PROGRAM INTERNAL PRG_TEST_FB_MANUALCONTROLLER
VAR
	bEnableTests : BOOL;

	bInitDone 			: BOOL;
	fbManualController 	: FB_ManualController;
	fbDevValve 			: FB_DevValve;
END_VAR

IF bEnableTests THEN
	IF NOT bInitDone THEN
		bInitDone := TRUE;
		fbDevValve.Init(
			nId := 1,
			nParentId := 0,
			eResetState := E_ValveResetState.Res_Idle,
			eSafeState := E_ValveResetState.Res_Idle
		);
	END_IF
	
	fbManualController();
	fbDevValve(
		refFbManualCtrl	:= fbManualController,
	);
END_IF

END_PROGRAM

(* stored: Version 1.1.0.1, ProductVersion 3.1.4024.11
   POU PRG_TEST_FB_MANUALCONTROLLER: Id {d21772fb-f5fd-0bd7-23c5-bca9237219d9}, SpecialFunc None *)
